FUNCTION_BLOCK FB_Axis_Continuous_NoHoming EXTENDS FB_Axis_NoHoming IMPLEMENTS ITF_Axis_Continuous
VAR_INPUT
END_VAR
VAR_OUTPUT
END_VAR
VAR
	//Internal Property Variables
	fModuloPosition		: LREAL;
	fModuloFactor		: LREAL;
END_VAR

PROPERTY ModuloFactor : LREAL
GET
ModuloFactor := fModuloFactor;
END_GET
END_PROPERTY

PROPERTY ModuloPosition : LREAL
GET
ModuloPosition := fModuloPosition;
END_GET
END_PROPERTY

METHOD Monitoring : BOOL
SUPER^.Monitoring();

fModuloPosition := SelectedAxis.NcToPlc.ModuloActPos;

IF fbWriteParameter.Done AND fbWriteParameter.ParameterNumber = MC_AxisParameter.AxisEncoderModuloValue THEN
	fModuloFactor := fbWriteParameter.Value;
END_IF

IF fbWriteParameter.Error AND NOT fbAxisBaseAlarms[E_AxisBase.WriteParameterError].bRaised THEN
	bError := TRUE;
	nErrorID := E_AxisBase.WriteParameterError;
	sTemp := UDINT_TO_STRING(fbWriteParameter.ErrorID);
	fbAxisBaseAlarms[E_AxisBase.WriteParameterError].ipArguments.Clear().AddString(sName).AddString(sTemp);
	fbAxisBaseAlarms[E_AxisBase.WriteParameterError].Raise(0);
ELSIF NOT fbAxisPower.Error AND fbAxisBaseAlarms[E_AxisBase.WriteParameterError].bRaised THEN
	fbAxisBaseAlarms[E_AxisBase.WriteParameterError].Clear(0,0);
END_IF
END_METHOD

METHOD SetAxisModuloFactor : BOOL
VAR_INPUT
	fSetAxisModuloFactor		: LREAL;
END_VAR
IF NOT bActive THEN
	IF NOT fbWriteParameter.Busy THEN
	fbWriteParameter(
						Axis:= SelectedAxis, 
						Execute:= TRUE, 
						ParameterNumber:= MC_AxisParameter.AxisEncoderModuloValue, 
						Value:= fSetAxisModuloFactor, 
						Done=> , 
						Busy=> , 
						Error=> , 
						ErrorID=> );
	END_IF
ELSE
	//TODO: Messaging for "Axis not ready for parameter write"
END_IF
END_METHOD

END_FUNCTION_BLOCK

(* stored: Version 1.1.0.1, ProductVersion 3.1.4024.9
   POU FB_Axis_Continuous_NoHoming: Id {5d6b6e86-fd8c-4cf5-a861-626e3257e9fc}, SpecialFunc None
   Folder 01_SUPER_Overrides: Id {fd7d4086-c0c0-4af3-8515-fa257fab9466}
   Folder 02_ITF_Axis_Continuous: Id {98dbdf85-b038-4db1-bbb7-5a2618f76ef7}
   Property ModuloFactor: Id {43ceaabc-2861-4ebd-867d-f031a89a2f60}
   Get Get: Id {6cda0ddf-c0d8-4a0e-bf9a-8414a9a42011}
   Property ModuloPosition: Id {c54c6b02-84af-4978-943b-973fa913e30f}
   Get Get: Id {5f0f54ee-1608-4fb3-819e-21c4e3d813ec}
   Method Monitoring: Id {2293e2b3-2922-4385-8328-b7feb57dcc0f}
   Method SetAxisModuloFactor: Id {3c4eda09-39c4-47ba-838e-d23f053f3a3d} *)
